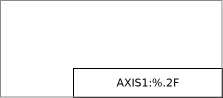
VISUALIZATION HMI  // 223x98
    Rectangle (73,68 150x30), "AXIS1:%.2F", text variable: MAIN.AXIS1.NcToPlc.ActPos
END_VISUALIZATION

(* stored: Version 1.1.0.1, ProductVersion 3.1.4024.5
   Visu HMI: Id {fdd2c5ad-0e60-4687-b65d-9b82648e23f4} *)
